(* Logix 5000 project; controller cal1632 1756-L62 rev 16.20; software revision 16.05; part 4 of 61 *)
(* tags used below, declared in another part *)
   AFI : BOOL;
   FAULT : BOOL;
   HMI : BOOL;
   p01_dint_to_hmi : DINT[16];
   p01_param_heater_hl : REAL;
   p01_param_process_air_hl : REAL;
   p01_param_process_air_max : REAL;
   p01_param_temp_limit : REAL;
   p01r01 : routine;
   p01r02 : routine;
   p01r02_all_fans_stopped : BOOL;
   p01r02_batch_run_time : DINT;
   p01r02_batch_run_time_hrs : DINT;
   p01r02_ethernet_comm : DINT;
   p01r02_fault_exists : BOOL;
   p01r02_flash_bit : BOOL;
   p01r02_flash_timer_off : TIMER;
   p01r02_flash_timer_on : TIMER;
   p01r02_plc_faults : DINT;
   p01r02_plc_scan_time : DINT;
   p01r02_plc_scan_time_in_sec : REAL;
   p01r02_timer_batch : TIMER;
   p01r02_timer_fault : TIMER[25];
   p01r02_timer_half_second_off : TIMER;
   p01r02_timer_half_second_on : TIMER;
   p01r02_timer_second : TIMER[2];
   p01r02_timer_warning : TIMER[4];
   p01r02_unack_fault : BOOL;
   p01r02_unack_warning : BOOL;
   p01r02_vfd_comm_2 : DINT[50];
   p01r02_warnings_exists : BOOL;
   p01r03 : routine;
   p01r04 : routine;
   p01r05 : routine;
   p01r06 : routine;
   p01r07 : routine;
   p01r08 : routine;
   p01r09 : routine;
   p01r09_pb_global_reset : BOOL;
   p01r10 : routine;
   p01r11 : routine;
   p01r12 : routine;
   p01r13 : routine;
   p01r13_line_running : BOOL;
   p02_dint_from_hmi : hmi_dint;
   p11r31_request_auto_run : BOOL;
   p11r32_request_auto_run : BOOL;
   p12r31_request_auto_run : BOOL;
   p12r32_request_auto_run : BOOL;
   p13r31_request_auto_run : BOOL;
   p13r32_request_auto_run : BOOL;
   p23_do_enable_impreg_exhaust_fan : BOOL;
   p23r13_request_auto_run : BOOL;

PROGRAM P01_System   (* main routine R01_Main *)
VAR
   tmrFlash : TIMER[4] := ([0].PRE := 1000, [0].ACC := 300, [1].PRE := 1000, [2].PRE := 500, [2].ACC := 300, [3].PRE := 500);   // Flash Timer
END_VAR

ROUTINE R01_Main   (* ladder *)
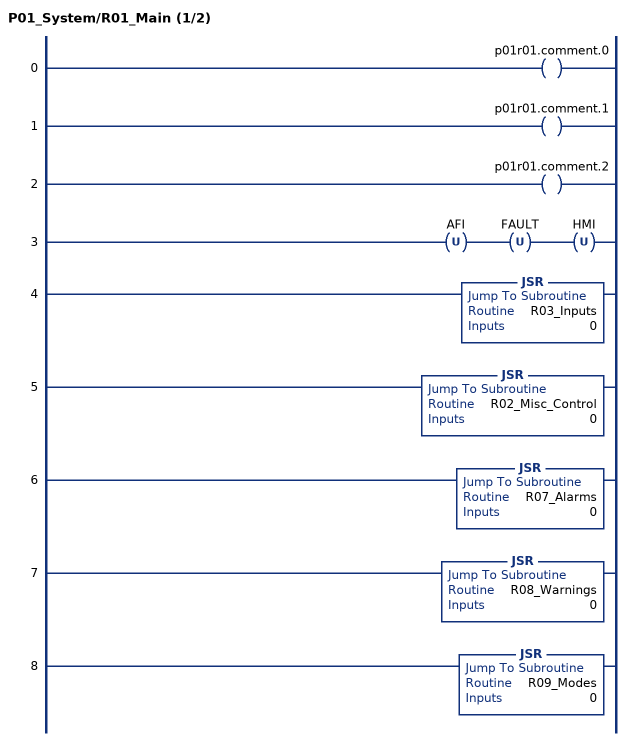
   0: OTE(p01r01.comment.0);
   1: OTE(p01r01.comment.1);
   2: OTE(p01r01.comment.2);
   3: OTU(AFI)OTU(FAULT)OTU(HMI);
   4: JSR(R03_Inputs,0);
   5: JSR(R02_Misc_Control,0);
   6: JSR(R07_Alarms,0);
   7: JSR(R08_Warnings,0);
   8: JSR(R09_Modes,0);
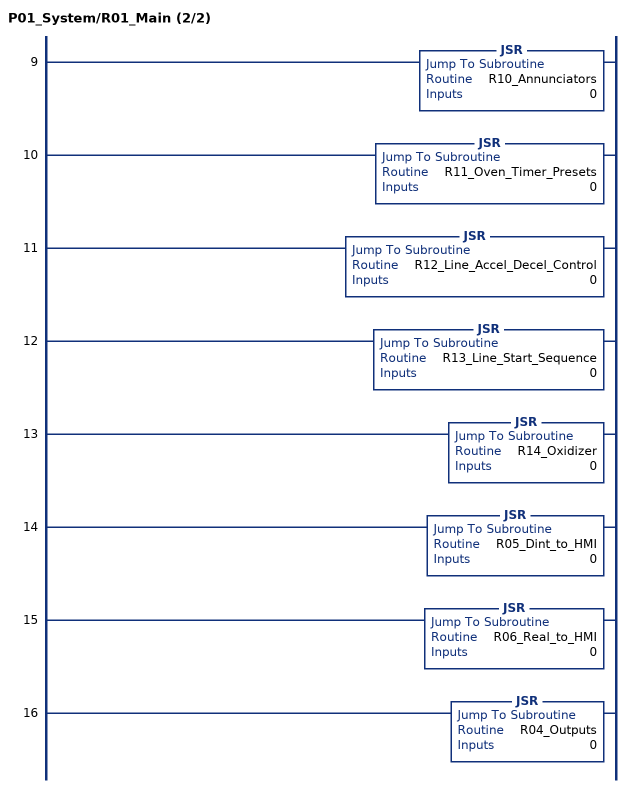
   9: JSR(R10_Annunciators,0);
   10: JSR(R11_Oven_Timer_Presets,0);
   11: JSR(R12_Line_Accel_Decel_Control,0);
   12: JSR(R13_Line_Start_Sequence,0);
   13: JSR(R14_Oxidizer,0);
   14: JSR(R05_Dint_to_HMI,0);
   15: JSR(R06_Real_to_HMI,0);
   16: JSR(R04_Outputs,0);
END_ROUTINE

ROUTINE R02_Misc_Control   (* ladder *)
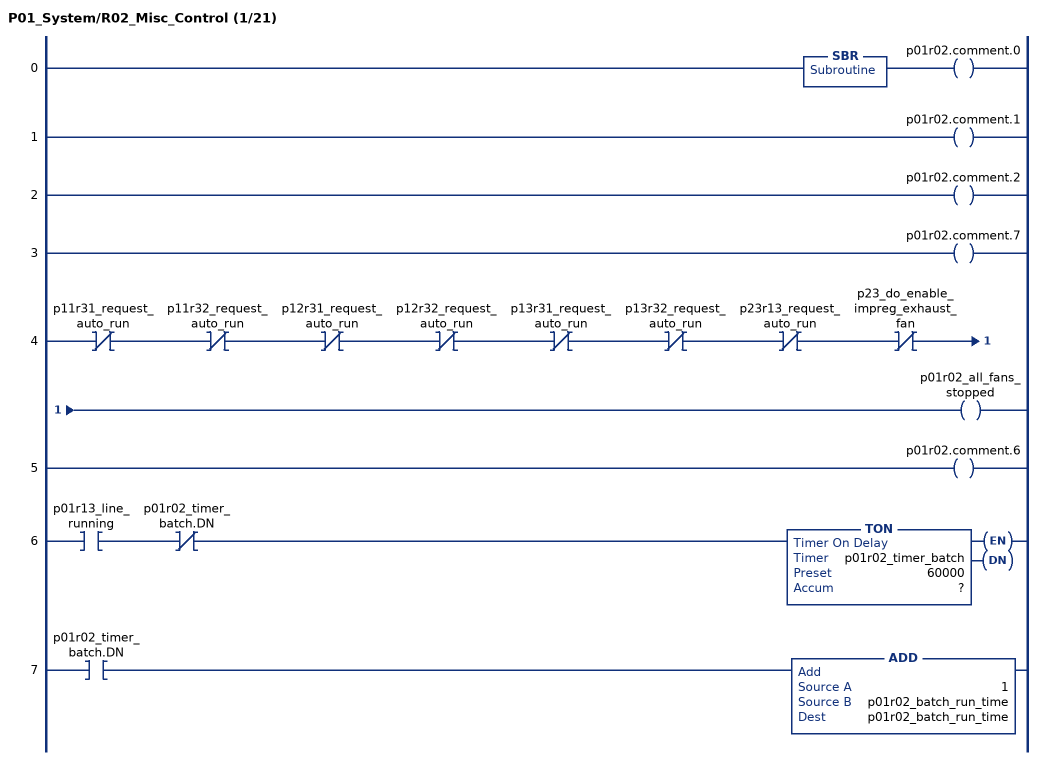
   0: SBR()OTE(p01r02.comment.0);
   1: OTE(p01r02.comment.1);
   2: OTE(p01r02.comment.2);
   3: OTE(p01r02.comment.7);
   4: XIO(p11r31_request_auto_run)XIO(p11r32_request_auto_run)XIO(p12r31_request_auto_run)XIO(p12r32_request_auto_run)XIO(p13r31_request_auto_run)XIO(p13r32_request_auto_run)XIO(p23r13_request_auto_run)XIO(p23_do_enable_impreg_exhaust_fan)OTE(p01r02_all_fans_stopped);
   5: OTE(p01r02.comment.6);
   6: XIC(p01r13_line_running)XIO(p01r02_timer_batch.DN)TON(p01r02_timer_batch,?,?);
   7: XIC(p01r02_timer_batch.DN)ADD(1,p01r02_batch_run_time,p01r02_batch_run_time);
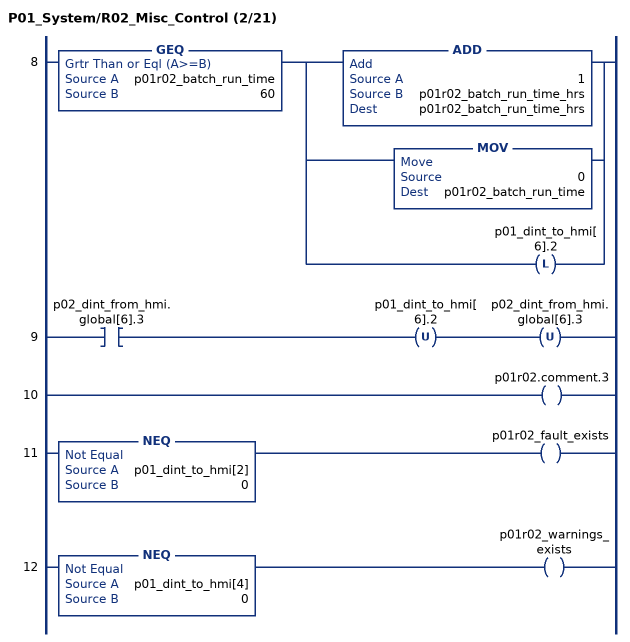
   8: GEQ(p01r02_batch_run_time,60)[ADD(1,p01r02_batch_run_time_hrs,p01r02_batch_run_time_hrs) ,MOV(0,p01r02_batch_run_time) ,OTL(p01_dint_to_hmi[6].2) ];
   9: XIC(p02_dint_from_hmi.global[6].3)OTU(p01_dint_to_hmi[6].2)OTU(p02_dint_from_hmi.global[6].3);
   10: OTE(p01r02.comment.3);
   11: NEQ(p01_dint_to_hmi[2],0)OTE(p01r02_fault_exists);
   12: NEQ(p01_dint_to_hmi[4],0)OTE(p01r02_warnings_exists);
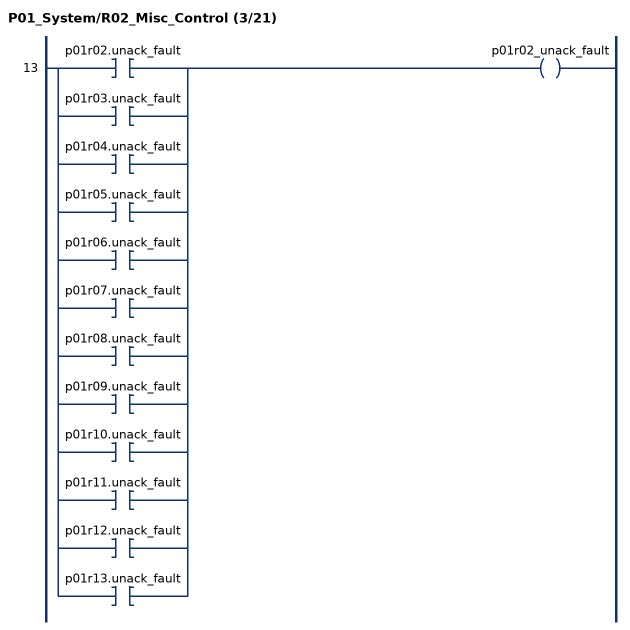
   13: [XIC(p01r02.unack_fault) ,XIC(p01r03.unack_fault) ,XIC(p01r04.unack_fault) ,XIC(p01r05.unack_fault) ,XIC(p01r06.unack_fault) ,XIC(p01r07.unack_fault) ,XIC(p01r08.unack_fault) ,XIC(p01r09.unack_fault) ,XIC(p01r10.unack_fault) ,XIC(p01r11.unack_fault) ,XIC(p01r12.unack_fault) ,XIC(p01r13.unack_fault) ]OTE(p01r02_unack_fault);
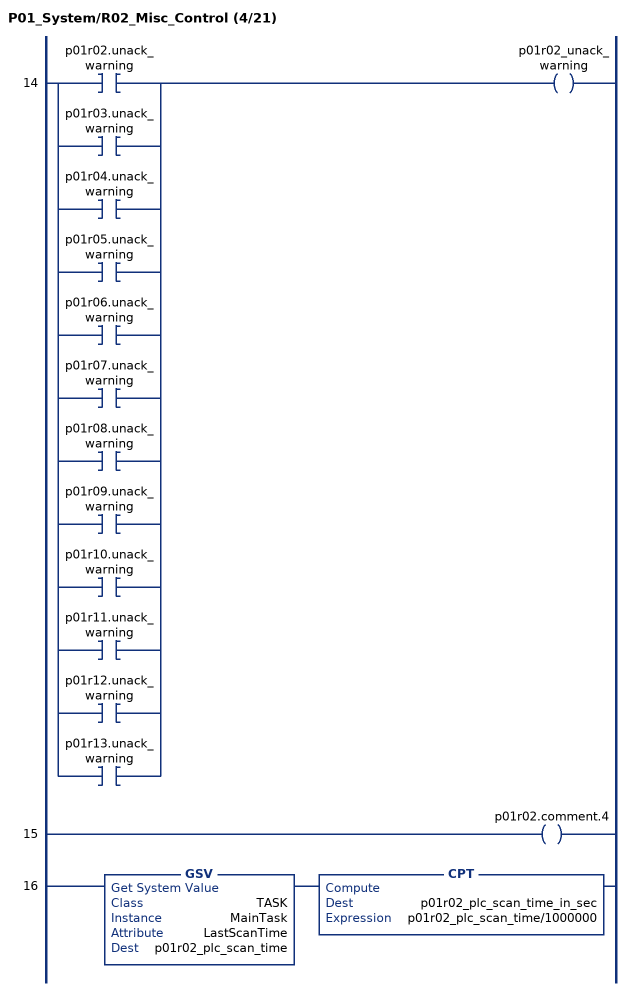
   14: [XIC(p01r02.unack_warning) ,XIC(p01r03.unack_warning) ,XIC(p01r04.unack_warning) ,XIC(p01r05.unack_warning) ,XIC(p01r06.unack_warning) ,XIC(p01r07.unack_warning) ,XIC(p01r08.unack_warning) ,XIC(p01r09.unack_warning) ,XIC(p01r10.unack_warning) ,XIC(p01r11.unack_warning) ,XIC(p01r12.unack_warning) ,XIC(p01r13.unack_warning) ]OTE(p01r02_unack_warning);
   15: OTE(p01r02.comment.4);
   16: GSV(TASK,MainTask,LastScanTime,p01r02_plc_scan_time)CPT(p01r02_plc_scan_time_in_sec,p01r02_plc_scan_time/1000000);
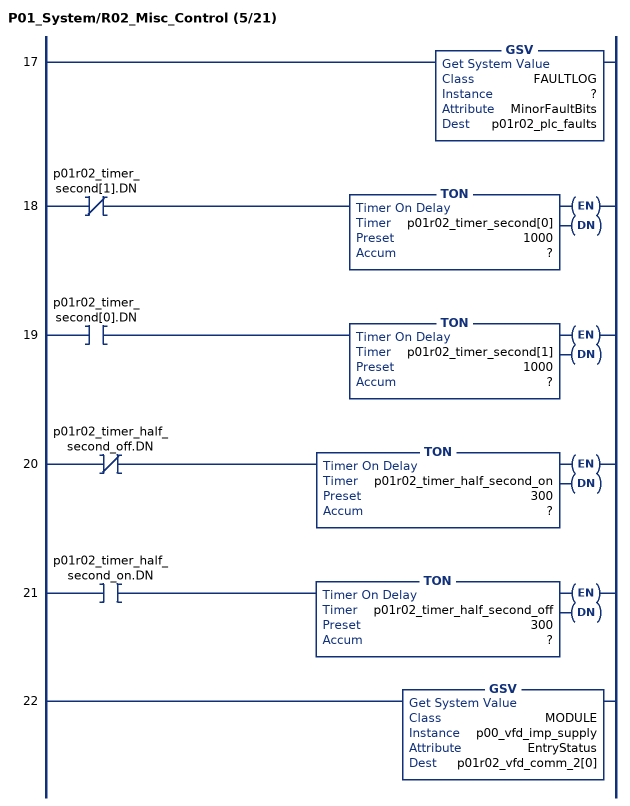
   17: GSV(FAULTLOG,?,MinorFaultBits,p01r02_plc_faults);
   18: XIO(p01r02_timer_second[1].DN)TON(p01r02_timer_second[0],?,?);
   19: XIC(p01r02_timer_second[0].DN)TON(p01r02_timer_second[1],?,?);
   20: XIO(p01r02_timer_half_second_off.DN)TON(p01r02_timer_half_second_on,?,?);
   21: XIC(p01r02_timer_half_second_on.DN)TON(p01r02_timer_half_second_off,?,?);
   22: GSV(MODULE,p00_vfd_imp_supply,EntryStatus,p01r02_vfd_comm_2[0]);
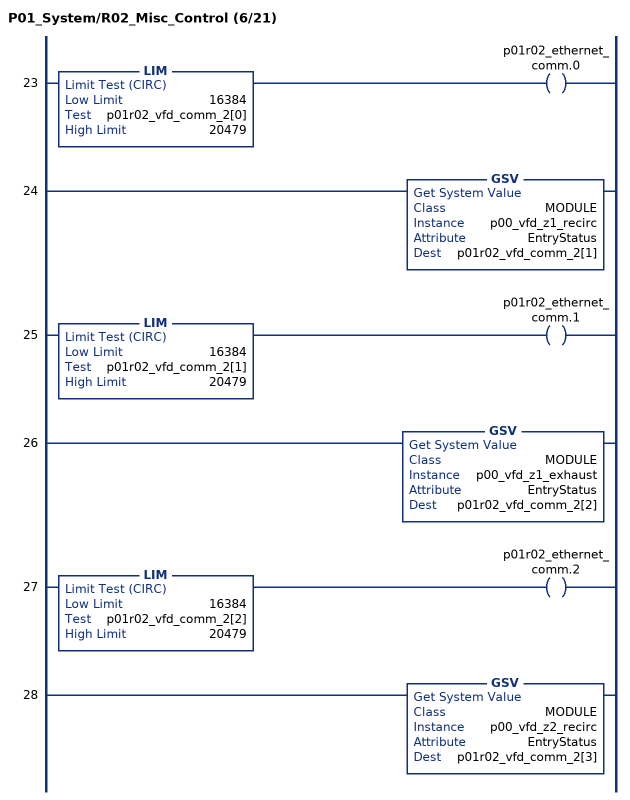
   23: LIM(16384,p01r02_vfd_comm_2[0],20479)OTE(p01r02_ethernet_comm.0);
   24: GSV(MODULE,p00_vfd_z1_recirc,EntryStatus,p01r02_vfd_comm_2[1]);
   25: LIM(16384,p01r02_vfd_comm_2[1],20479)OTE(p01r02_ethernet_comm.1);
   26: GSV(MODULE,p00_vfd_z1_exhaust,EntryStatus,p01r02_vfd_comm_2[2]);
   27: LIM(16384,p01r02_vfd_comm_2[2],20479)OTE(p01r02_ethernet_comm.2);
   28: GSV(MODULE,p00_vfd_z2_recirc,EntryStatus,p01r02_vfd_comm_2[3]);
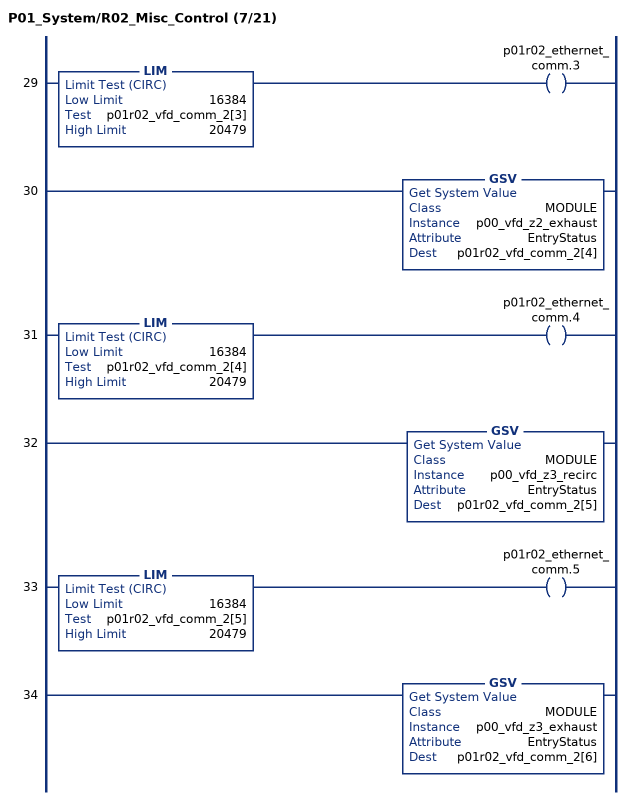
   29: LIM(16384,p01r02_vfd_comm_2[3],20479)OTE(p01r02_ethernet_comm.3);
   30: GSV(MODULE,p00_vfd_z2_exhaust,EntryStatus,p01r02_vfd_comm_2[4]);
   31: LIM(16384,p01r02_vfd_comm_2[4],20479)OTE(p01r02_ethernet_comm.4);
   32: GSV(MODULE,p00_vfd_z3_recirc,EntryStatus,p01r02_vfd_comm_2[5]);
   33: LIM(16384,p01r02_vfd_comm_2[5],20479)OTE(p01r02_ethernet_comm.5);
   34: GSV(MODULE,p00_vfd_z3_exhaust,EntryStatus,p01r02_vfd_comm_2[6]);
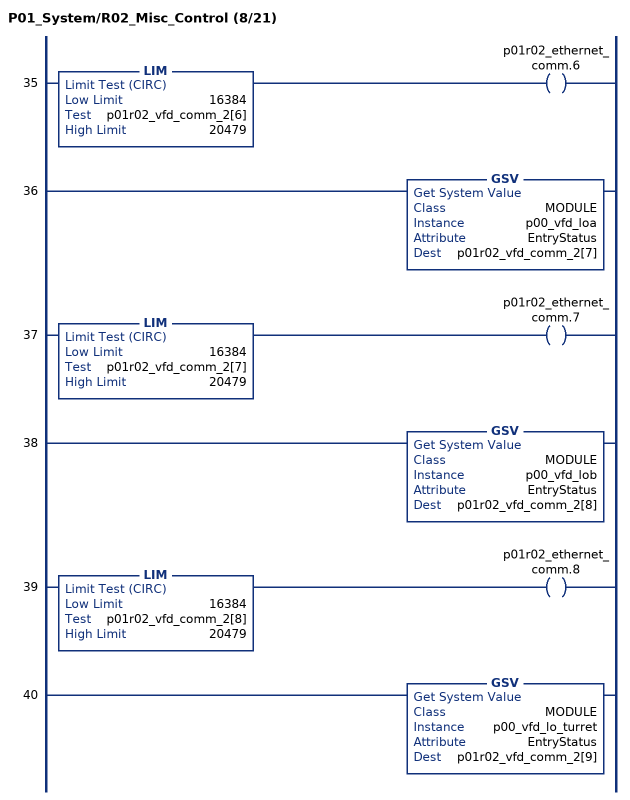
   35: LIM(16384,p01r02_vfd_comm_2[6],20479)OTE(p01r02_ethernet_comm.6);
   36: GSV(MODULE,p00_vfd_loa,EntryStatus,p01r02_vfd_comm_2[7]);
   37: LIM(16384,p01r02_vfd_comm_2[7],20479)OTE(p01r02_ethernet_comm.7);
   38: GSV(MODULE,p00_vfd_lob,EntryStatus,p01r02_vfd_comm_2[8]);
   39: LIM(16384,p01r02_vfd_comm_2[8],20479)OTE(p01r02_ethernet_comm.8);
   40: GSV(MODULE,p00_vfd_lo_turret,EntryStatus,p01r02_vfd_comm_2[9]);
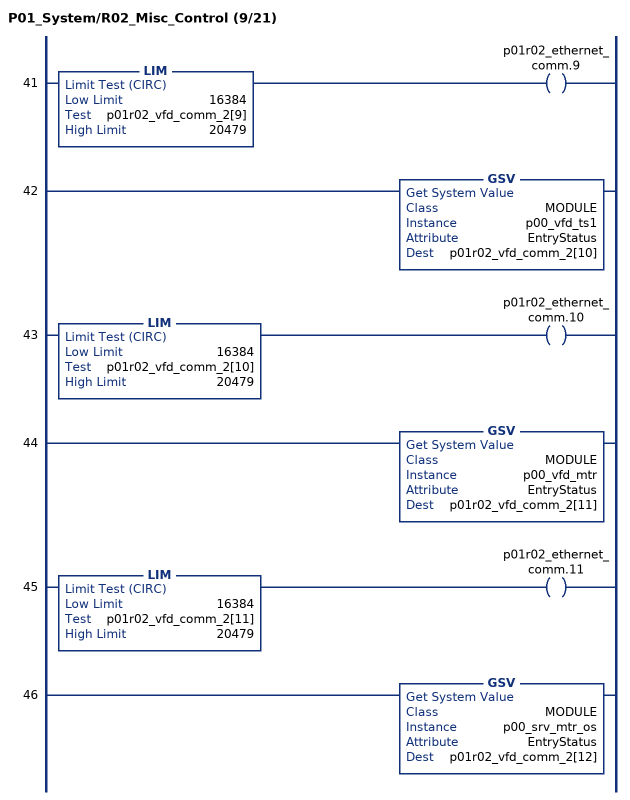
   41: LIM(16384,p01r02_vfd_comm_2[9],20479)OTE(p01r02_ethernet_comm.9);
   42: GSV(MODULE,p00_vfd_ts1,EntryStatus,p01r02_vfd_comm_2[10]);
   43: LIM(16384,p01r02_vfd_comm_2[10],20479)OTE(p01r02_ethernet_comm.10);
   44: GSV(MODULE,p00_vfd_mtr,EntryStatus,p01r02_vfd_comm_2[11]);
   45: LIM(16384,p01r02_vfd_comm_2[11],20479)OTE(p01r02_ethernet_comm.11);
   46: GSV(MODULE,p00_srv_mtr_os,EntryStatus,p01r02_vfd_comm_2[12]);
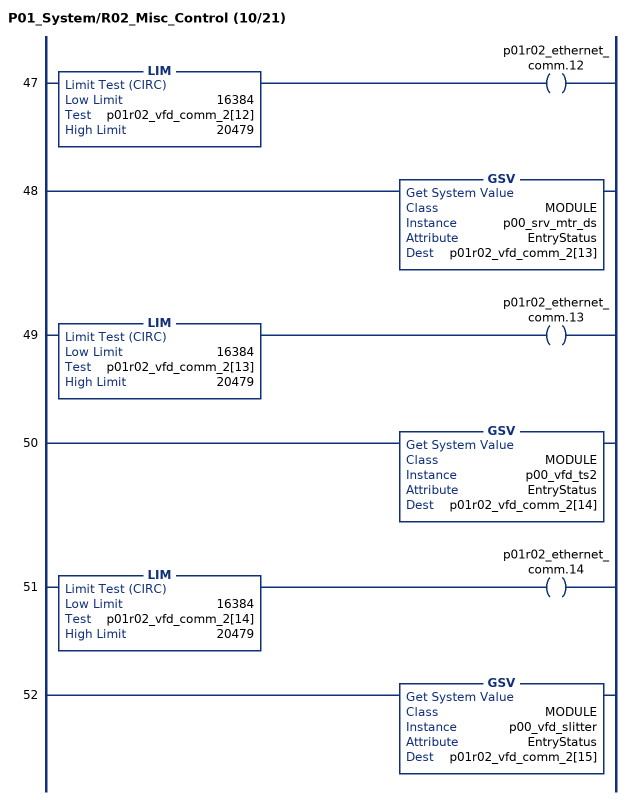
   47: LIM(16384,p01r02_vfd_comm_2[12],20479)OTE(p01r02_ethernet_comm.12);
   48: GSV(MODULE,p00_srv_mtr_ds,EntryStatus,p01r02_vfd_comm_2[13]);
   49: LIM(16384,p01r02_vfd_comm_2[13],20479)OTE(p01r02_ethernet_comm.13);
   50: GSV(MODULE,p00_vfd_ts2,EntryStatus,p01r02_vfd_comm_2[14]);
   51: LIM(16384,p01r02_vfd_comm_2[14],20479)OTE(p01r02_ethernet_comm.14);
   52: GSV(MODULE,p00_vfd_slitter,EntryStatus,p01r02_vfd_comm_2[15]);
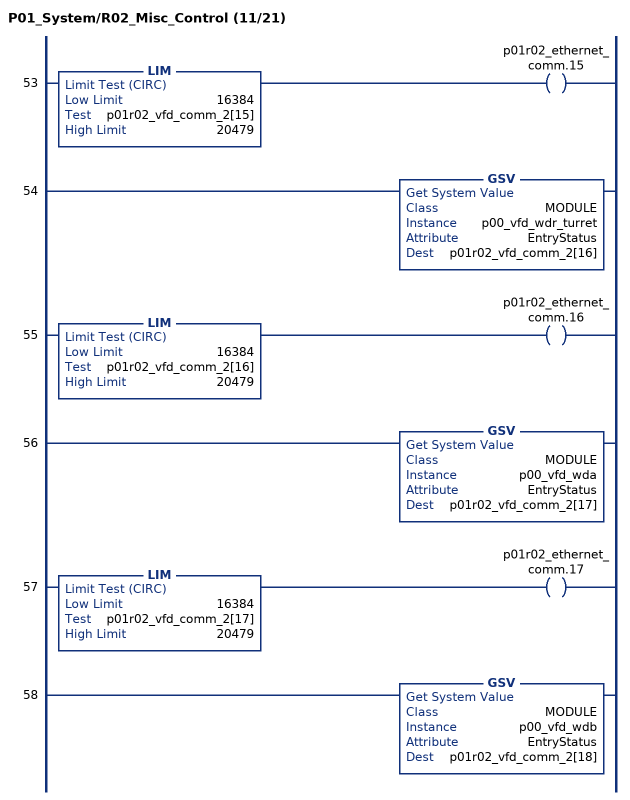
   53: LIM(16384,p01r02_vfd_comm_2[15],20479)OTE(p01r02_ethernet_comm.15);
   54: GSV(MODULE,p00_vfd_wdr_turret,EntryStatus,p01r02_vfd_comm_2[16]);
   55: LIM(16384,p01r02_vfd_comm_2[16],20479)OTE(p01r02_ethernet_comm.16);
   56: GSV(MODULE,p00_vfd_wda,EntryStatus,p01r02_vfd_comm_2[17]);
   57: LIM(16384,p01r02_vfd_comm_2[17],20479)OTE(p01r02_ethernet_comm.17);
   58: GSV(MODULE,p00_vfd_wdb,EntryStatus,p01r02_vfd_comm_2[18]);
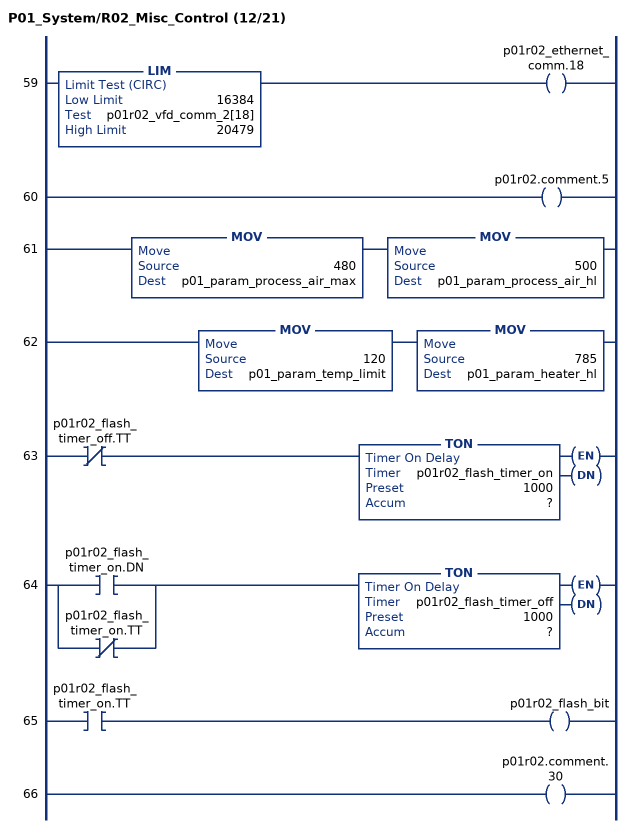
   59: LIM(16384,p01r02_vfd_comm_2[18],20479)OTE(p01r02_ethernet_comm.18);
   60: OTE(p01r02.comment.5);
   61: MOV(480,p01_param_process_air_max)MOV(500,p01_param_process_air_hl);
   62: MOV(120,p01_param_temp_limit)MOV(785,p01_param_heater_hl);
   63: XIO(p01r02_flash_timer_off.TT)TON(p01r02_flash_timer_on,?,?);
   64: [XIC(p01r02_flash_timer_on.DN) ,XIO(p01r02_flash_timer_on.TT) ]TON(p01r02_flash_timer_off,?,?);
   65: XIC(p01r02_flash_timer_on.TT)OTE(p01r02_flash_bit);
   66: OTE(p01r02.comment.30);
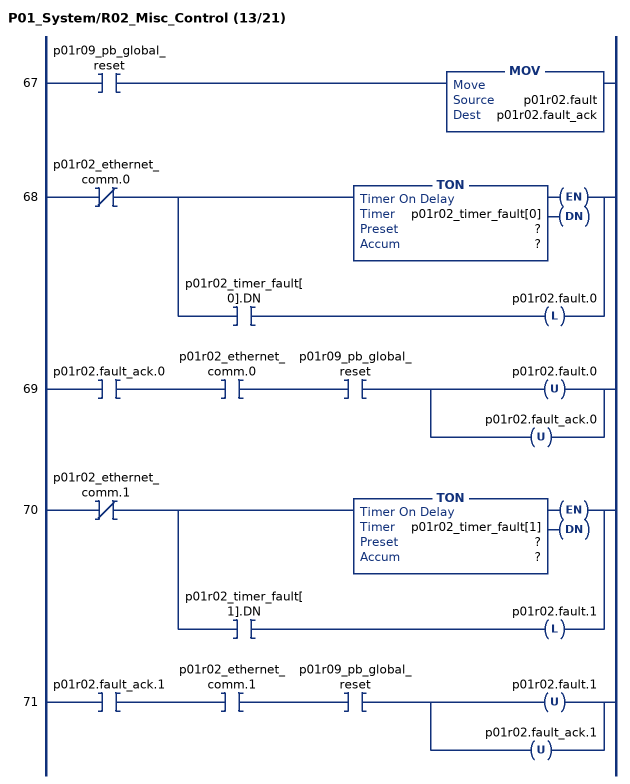
   67: XIC(p01r09_pb_global_reset)MOV(p01r02.fault,p01r02.fault_ack);
   68: XIO(p01r02_ethernet_comm.0)[TON(p01r02_timer_fault[0],?,?) ,XIC(p01r02_timer_fault[0].DN) OTL(p01r02.fault.0) ];
   69: XIC(p01r02.fault_ack.0)XIC(p01r02_ethernet_comm.0)XIC(p01r09_pb_global_reset)[OTU(p01r02.fault.0) ,OTU(p01r02.fault_ack.0) ];
   70: XIO(p01r02_ethernet_comm.1)[TON(p01r02_timer_fault[1],?,?) ,XIC(p01r02_timer_fault[1].DN) OTL(p01r02.fault.1) ];
   71: XIC(p01r02.fault_ack.1)XIC(p01r02_ethernet_comm.1)XIC(p01r09_pb_global_reset)[OTU(p01r02.fault.1) ,OTU(p01r02.fault_ack.1) ];
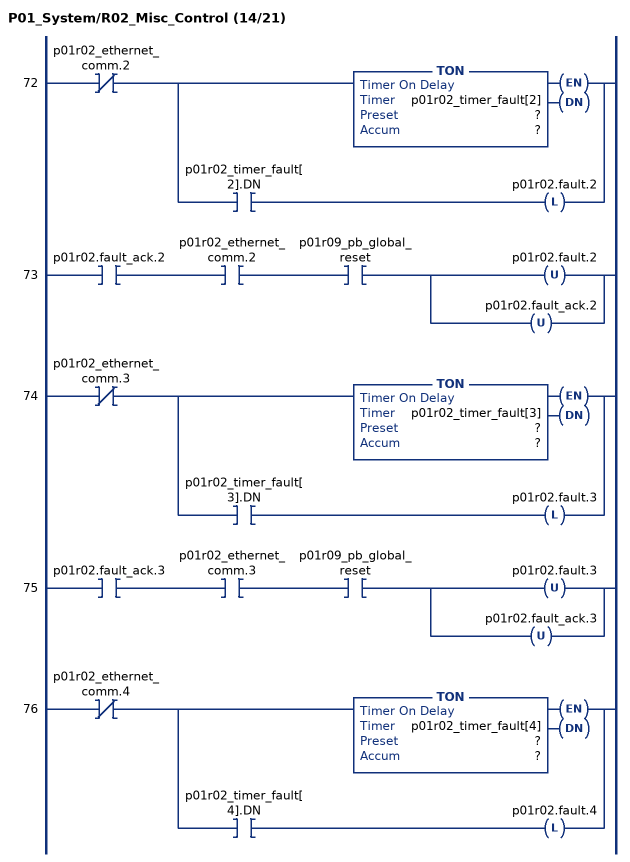
   72: XIO(p01r02_ethernet_comm.2)[TON(p01r02_timer_fault[2],?,?) ,XIC(p01r02_timer_fault[2].DN) OTL(p01r02.fault.2) ];
   73: XIC(p01r02.fault_ack.2)XIC(p01r02_ethernet_comm.2)XIC(p01r09_pb_global_reset)[OTU(p01r02.fault.2) ,OTU(p01r02.fault_ack.2) ];
   74: XIO(p01r02_ethernet_comm.3)[TON(p01r02_timer_fault[3],?,?) ,XIC(p01r02_timer_fault[3].DN) OTL(p01r02.fault.3) ];
   75: XIC(p01r02.fault_ack.3)XIC(p01r02_ethernet_comm.3)XIC(p01r09_pb_global_reset)[OTU(p01r02.fault.3) ,OTU(p01r02.fault_ack.3) ];
   76: XIO(p01r02_ethernet_comm.4)[TON(p01r02_timer_fault[4],?,?) ,XIC(p01r02_timer_fault[4].DN) OTL(p01r02.fault.4) ];
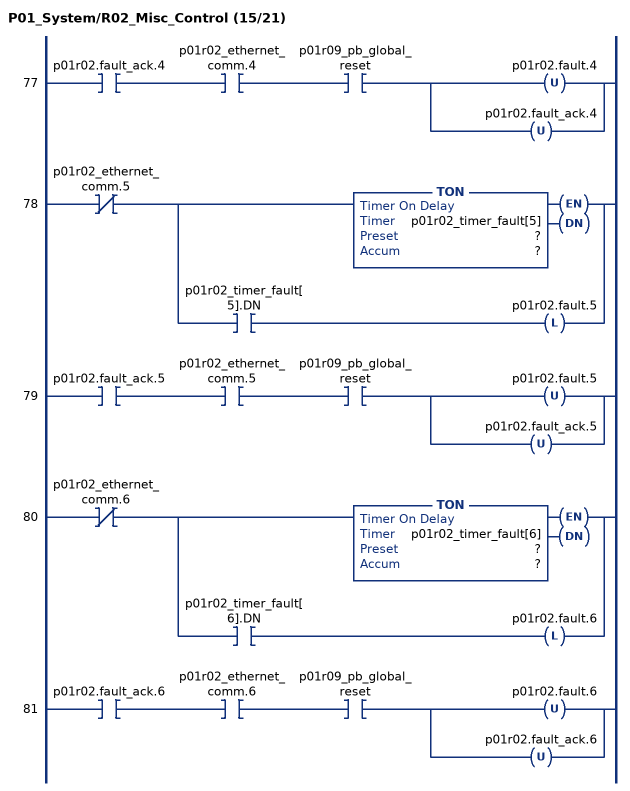
   77: XIC(p01r02.fault_ack.4)XIC(p01r02_ethernet_comm.4)XIC(p01r09_pb_global_reset)[OTU(p01r02.fault.4) ,OTU(p01r02.fault_ack.4) ];
   78: XIO(p01r02_ethernet_comm.5)[TON(p01r02_timer_fault[5],?,?) ,XIC(p01r02_timer_fault[5].DN) OTL(p01r02.fault.5) ];
   79: XIC(p01r02.fault_ack.5)XIC(p01r02_ethernet_comm.5)XIC(p01r09_pb_global_reset)[OTU(p01r02.fault.5) ,OTU(p01r02.fault_ack.5) ];
   80: XIO(p01r02_ethernet_comm.6)[TON(p01r02_timer_fault[6],?,?) ,XIC(p01r02_timer_fault[6].DN) OTL(p01r02.fault.6) ];
   81: XIC(p01r02.fault_ack.6)XIC(p01r02_ethernet_comm.6)XIC(p01r09_pb_global_reset)[OTU(p01r02.fault.6) ,OTU(p01r02.fault_ack.6) ];
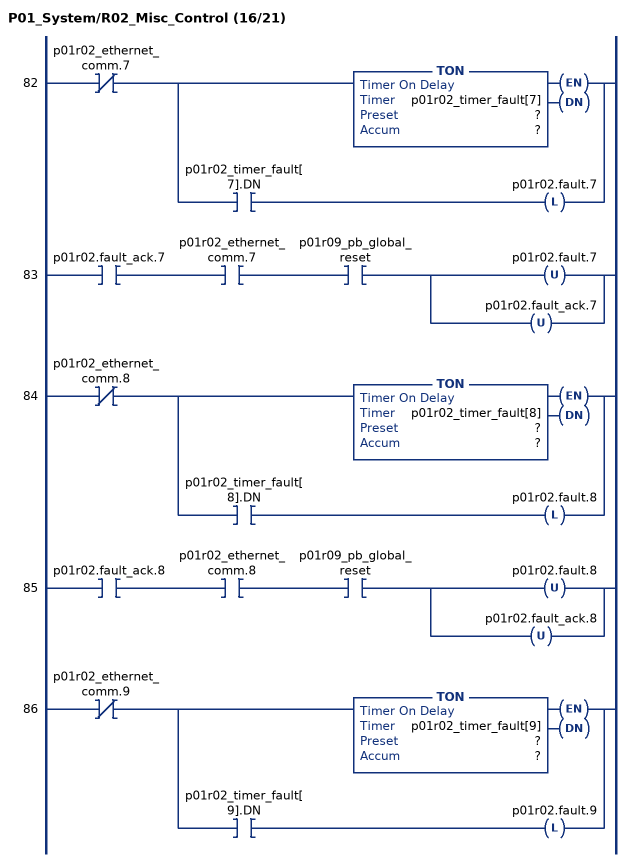
   82: XIO(p01r02_ethernet_comm.7)[TON(p01r02_timer_fault[7],?,?) ,XIC(p01r02_timer_fault[7].DN) OTL(p01r02.fault.7) ];
   83: XIC(p01r02.fault_ack.7)XIC(p01r02_ethernet_comm.7)XIC(p01r09_pb_global_reset)[OTU(p01r02.fault.7) ,OTU(p01r02.fault_ack.7) ];
   84: XIO(p01r02_ethernet_comm.8)[TON(p01r02_timer_fault[8],?,?) ,XIC(p01r02_timer_fault[8].DN) OTL(p01r02.fault.8) ];
   85: XIC(p01r02.fault_ack.8)XIC(p01r02_ethernet_comm.8)XIC(p01r09_pb_global_reset)[OTU(p01r02.fault.8) ,OTU(p01r02.fault_ack.8) ];
   86: XIO(p01r02_ethernet_comm.9)[TON(p01r02_timer_fault[9],?,?) ,XIC(p01r02_timer_fault[9].DN) OTL(p01r02.fault.9) ];
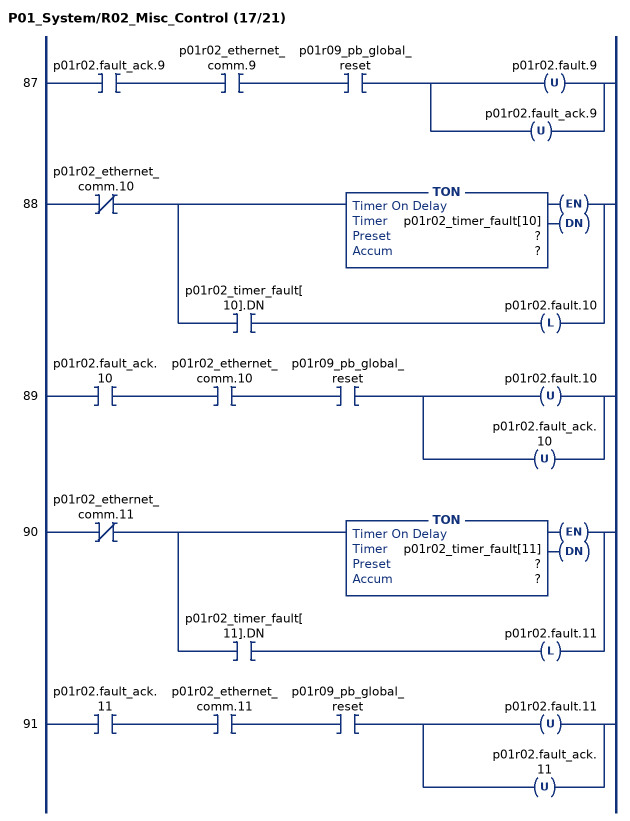
   87: XIC(p01r02.fault_ack.9)XIC(p01r02_ethernet_comm.9)XIC(p01r09_pb_global_reset)[OTU(p01r02.fault.9) ,OTU(p01r02.fault_ack.9) ];
   88: XIO(p01r02_ethernet_comm.10)[TON(p01r02_timer_fault[10],?,?) ,XIC(p01r02_timer_fault[10].DN) OTL(p01r02.fault.10) ];
   89: XIC(p01r02.fault_ack.10)XIC(p01r02_ethernet_comm.10)XIC(p01r09_pb_global_reset)[OTU(p01r02.fault.10) ,OTU(p01r02.fault_ack.10) ];
   90: XIO(p01r02_ethernet_comm.11)[TON(p01r02_timer_fault[11],?,?) ,XIC(p01r02_timer_fault[11].DN) OTL(p01r02.fault.11) ];
   91: XIC(p01r02.fault_ack.11)XIC(p01r02_ethernet_comm.11)XIC(p01r09_pb_global_reset)[OTU(p01r02.fault.11) ,OTU(p01r02.fault_ack.11) ];
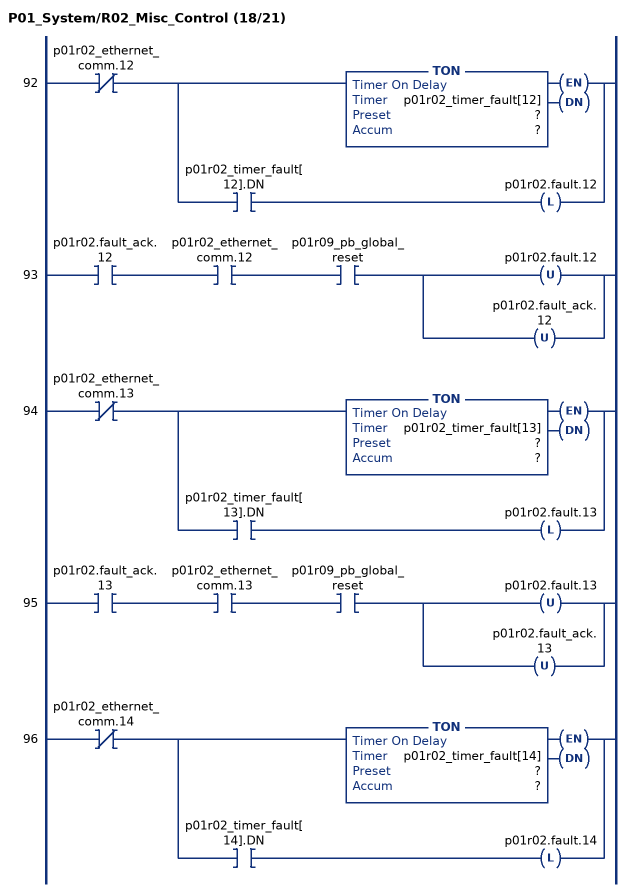
   92: XIO(p01r02_ethernet_comm.12)[TON(p01r02_timer_fault[12],?,?) ,XIC(p01r02_timer_fault[12].DN) OTL(p01r02.fault.12) ];
   93: XIC(p01r02.fault_ack.12)XIC(p01r02_ethernet_comm.12)XIC(p01r09_pb_global_reset)[OTU(p01r02.fault.12) ,OTU(p01r02.fault_ack.12) ];
   94: XIO(p01r02_ethernet_comm.13)[TON(p01r02_timer_fault[13],?,?) ,XIC(p01r02_timer_fault[13].DN) OTL(p01r02.fault.13) ];
   95: XIC(p01r02.fault_ack.13)XIC(p01r02_ethernet_comm.13)XIC(p01r09_pb_global_reset)[OTU(p01r02.fault.13) ,OTU(p01r02.fault_ack.13) ];
   96: XIO(p01r02_ethernet_comm.14)[TON(p01r02_timer_fault[14],?,?) ,XIC(p01r02_timer_fault[14].DN) OTL(p01r02.fault.14) ];
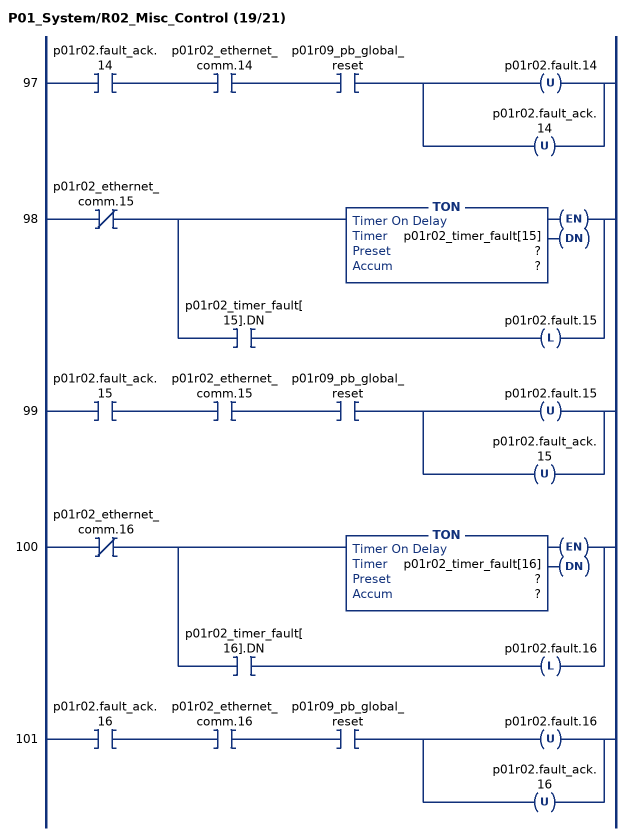
   97: XIC(p01r02.fault_ack.14)XIC(p01r02_ethernet_comm.14)XIC(p01r09_pb_global_reset)[OTU(p01r02.fault.14) ,OTU(p01r02.fault_ack.14) ];
   98: XIO(p01r02_ethernet_comm.15)[TON(p01r02_timer_fault[15],?,?) ,XIC(p01r02_timer_fault[15].DN) OTL(p01r02.fault.15) ];
   99: XIC(p01r02.fault_ack.15)XIC(p01r02_ethernet_comm.15)XIC(p01r09_pb_global_reset)[OTU(p01r02.fault.15) ,OTU(p01r02.fault_ack.15) ];
   100: XIO(p01r02_ethernet_comm.16)[TON(p01r02_timer_fault[16],?,?) ,XIC(p01r02_timer_fault[16].DN) OTL(p01r02.fault.16) ];
   101: XIC(p01r02.fault_ack.16)XIC(p01r02_ethernet_comm.16)XIC(p01r09_pb_global_reset)[OTU(p01r02.fault.16) ,OTU(p01r02.fault_ack.16) ];
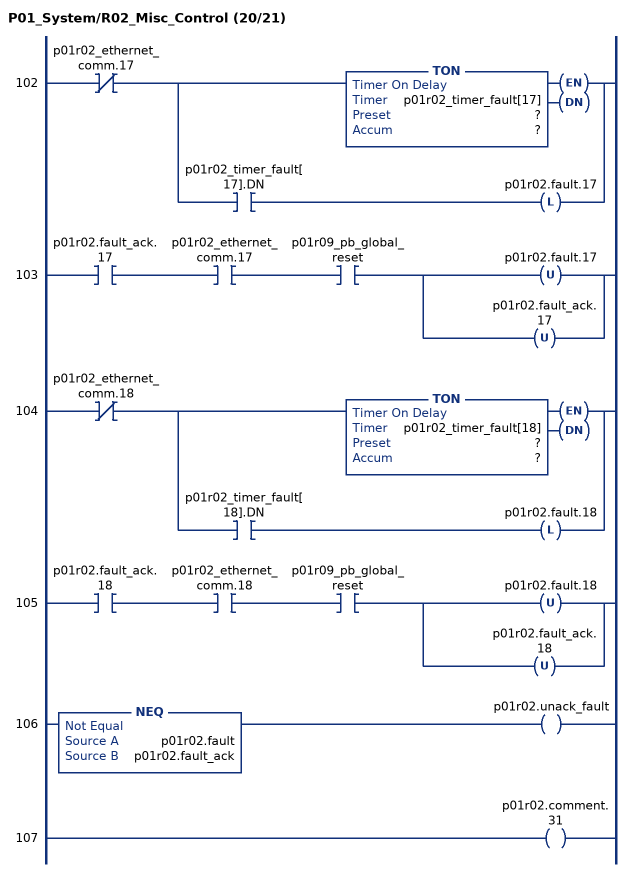
   102: XIO(p01r02_ethernet_comm.17)[TON(p01r02_timer_fault[17],?,?) ,XIC(p01r02_timer_fault[17].DN) OTL(p01r02.fault.17) ];
   103: XIC(p01r02.fault_ack.17)XIC(p01r02_ethernet_comm.17)XIC(p01r09_pb_global_reset)[OTU(p01r02.fault.17) ,OTU(p01r02.fault_ack.17) ];
   104: XIO(p01r02_ethernet_comm.18)[TON(p01r02_timer_fault[18],?,?) ,XIC(p01r02_timer_fault[18].DN) OTL(p01r02.fault.18) ];
   105: XIC(p01r02.fault_ack.18)XIC(p01r02_ethernet_comm.18)XIC(p01r09_pb_global_reset)[OTU(p01r02.fault.18) ,OTU(p01r02.fault_ack.18) ];
   106: NEQ(p01r02.fault,p01r02.fault_ack)OTE(p01r02.unack_fault);
   107: OTE(p01r02.comment.31);
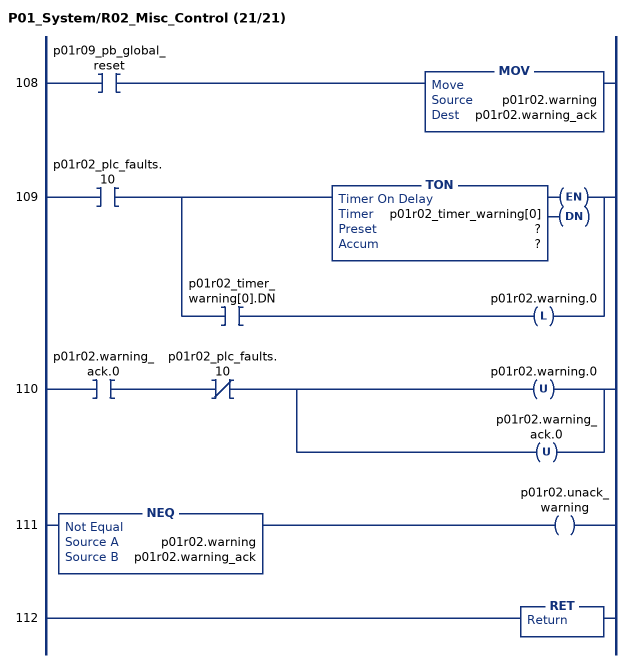
   108: XIC(p01r09_pb_global_reset)MOV(p01r02.warning,p01r02.warning_ack);
   109: XIC(p01r02_plc_faults.10)[TON(p01r02_timer_warning[0],?,?) ,XIC(p01r02_timer_warning[0].DN) OTL(p01r02.warning.0) ];
   110: XIC(p01r02.warning_ack.0)XIO(p01r02_plc_faults.10)[OTU(p01r02.warning.0) ,OTU(p01r02.warning_ack.0) ];
   111: NEQ(p01r02.warning,p01r02.warning_ack)OTE(p01r02.unack_warning);
   112: RET();
END_ROUTINE
